PROGRAM ControlTemp
VAR
	FB_CTRL_TempControllerTop: FB_CTRL_TempController;
	FB_CTRL_TempControllerBot: FB_CTRL_TempController;
	modo:E_CTRL_MODE:=eCTRL_MODE_ACTIVE;
	
	sControllerParameter: ST_CTRL_TempCtrlParameter:=
	(
			(* general parameters *)
			iMode                     :=1,
			bSelCtrlParameterSet      :=TRUE,
			tCtrlCycleTime            :=T#100MS,
			tTaskCycleTime            :=T#10MS,

		  (* tuning parameteer *)
		  iTuningMode               := eCTRL_TuneMode_HEATING,
		  tTuneStabilisation        := T#30S,
		  fEndTunePercentHeating    := 80.0,
		  fYTuneHeating:=100.0,
		  fEndTunePercentCooling    := 20.0,
		  fYStableCooling:=50.0,
		  fScalingFactor            := 1.0,
		
		  (* setpoint parameters *)
		  fWMin:=0.0,
		  fWMax:=573.0,

		  (* start up *)
		  bEnableSoftStart:=FALSE,
		  bEnableRamping:=TRUE,
		  fWStartUp:=348.0,
		  tStartUp:=T#30S,
		  bStartUpRamping:=TRUE,
		  fWStartUpVeloPos:=3.0,
		  fWStartUpVeloNeg:=3.0,
		  fWVeloPos:=5.0,
		  fWVeloNeg:=5.0,
		
		  (* actual value parameters *)
		  bFilter:=FALSE,
		  tFilter:=T#100MS,
		
		  (* deadband parameters *)
		  bDeadband:=FALSE,
		  fEDeadband:=1.0,
		  
		  (* control value parameters *)
		  fYMin:=0.0,
		  fYMax:=573.0,
		  fYManual:=20.0,
		  fYOnFailure:=20.0,
		  tPWMCycleTime:=T#100MS,
		  tPWMMinOffTime:=T#100MS,
		  tPWMMinOnTime:=T#100MS,
		  tPWMWaitingTime:=T#100MS,
		  fYThresholdOff:=50.0,
		  fYThresholdOn:=50.0,
		  nCyclesForSwitchOver      := 100,
		
		  (* controller settings *)
		  bEnablePreController:=FALSE,
		  bEnableZones:=FALSE,
		  bEnableCVFilter:=FALSE,
		  iFilterType:=eCTRL_FilterType_AVERAGE,
		  iControllerType:=eCTRL_ControllerType_PID,
		
		  (* min max temperatures *)
		  TempLow:=283.0,
		  TempLowLow:=0.0,
		  TempHigh:=503.0,
		  TempHighHigh:=523.0,
		  TempAbsoluteHigh:=523.0,
		  TempAbsoluteLow:=0.0,
		
		  (* internal tuning parameters *)
		  fTuneKp                   := 1.2,
		  fTuneTn                   := 2.0,
		  fTuneTv                   := 0.42,
		  fTuneTd                   := 0.25
  );
		
	//sControllerParameter
	sControllerParameter2:ST_CTRL_TempCtrlParameter:=
	(
		(* base *)
		tCtrlCycleTime := T#1000MS,
		tTaskCycleTime := T#10MS,
		
		fYMin := -100,
		fYMax := 100,
		tPWMCycleTime := T#100MS ,
		fYManual := 20,
		bFilter := FALSE,
		tFilter := T#100MS,
		bDeadband := FALSE,
		fEDeadband := 1.0, (* deadband *)
		fWMin := 288,
		fWMax := 523,
		fWStartUp := 323,
		tStartUp := T#1S,
		fWVeloPos := 0.5,
		fWVeloNeg := 0.5,
		bStartUpRamping := TRUE,
		fWStartUpVeloPos := 0.5,
		fWStartUpVeloNeg := 0.5,
		iMode := eCTRL_ControlMode_HEATING,
		dwAlarmSupp := 16#FF_FF_FF_FF,
		bSelCtrlParameterSet:= FALSE,
		
		(* tuninig *)
		iTuningMode := eCTRL_TuneMode_heating,
		fYTuneHeating := 100.0,
		fYTuneCooling := -100.0,
		fEndTunePercentHeating := 80.0, (* switch to closed loop control when X > 0.8*W *)
		fEndTunePercentCooling := -70.0, (* switch to closed loop control when X < 0.2*W *)
		iReactionOnFailure := eCTRL_ReactionOnFailure_StopController,
		TempLow := -50.0,
		TempLowLow := -100.0,
		TempHigh := 523,
		TempHighHigh := 523,
		TempAbsoluteHigh := 523,
		TempAbsoluteLow := -95.0,
		bEnablePreController := FALSE,
		bEnableZones := FALSE,
		bEnableCVFilter := FALSE,
		iFilterType := eCTRL_FilterType_AVERAGE,
		iControllerType := eCTRL_ControllerType_PID
	);
END_VAR

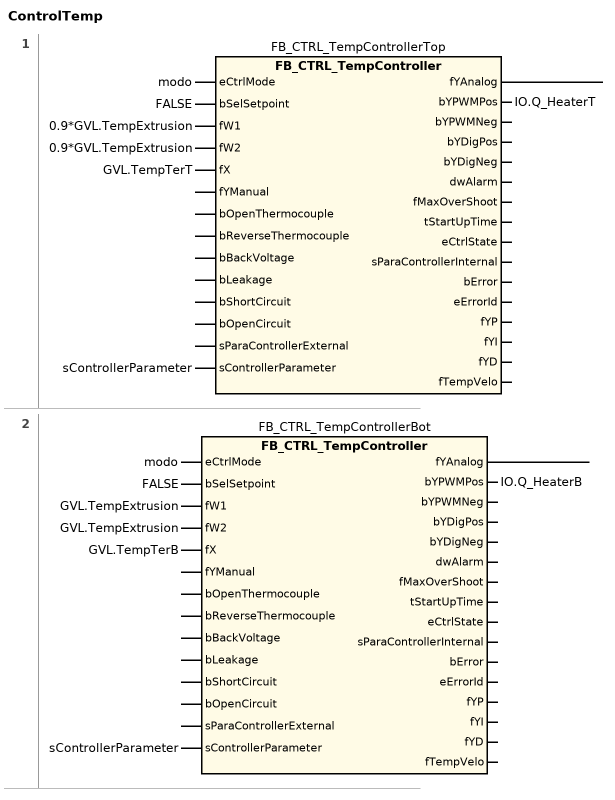
// NETWORK 1
FB_CTRL_TempControllerTop(
    eCtrlMode := modo,
    bSelSetpoint := FALSE,
    fW1 := 0.9*GVL.TempExtrusion,
    fW2 := 0.9*GVL.TempExtrusion,
    fX := GVL.TempTerT,
    sControllerParameter := sControllerParameter,
    bYPWMPos => IO.Q_HeaterT); // FB_CTRL_TempController

// NETWORK 2
FB_CTRL_TempControllerBot(
    eCtrlMode := modo,
    bSelSetpoint := FALSE,
    fW1 := GVL.TempExtrusion,
    fW2 := GVL.TempExtrusion,
    fX := GVL.TempTerB,
    sControllerParameter := sControllerParameter,
    bYPWMPos => IO.Q_HeaterB); // FB_CTRL_TempController

END_PROGRAM

(* stored: Version 1.1.0.1, ProductVersion 3.1.4024.9
   POU ControlTemp: Id {0e8e534b-cf5f-4841-8555-305e5ee6bfa8}, SpecialFunc None *)
